// TIA Portal V16 export
// export: Created 2021-09-01T08:19:45.6334848Z, ExportSetting WithDefaults, DisplayName Totally Integrated Automation Portal, DisplayVersion V16 Update 3, DisplayName TIA Portal Version Control Interface, DisplayVersion V16 Update 2, DisplayName TIA Portal Openness, DisplayVersion V16 Update 3, DisplayName TIA Portal Teamcenter Gateway, DisplayVersion V16, DisplayName STEP 7 Professional, DisplayVersion V16 Update 3, DisplayName STEP 7 Safety, DisplayVersion V16, DisplayName WinCC Advanced, DisplayVersion V16 Update 3
TYPE "SeqStep"
// stored: IsFailsafeCompliant false
   STRUCT
      StepDev { S7_SetPoint := 'True'} : Array[1..32] of Word;
      StepDelay { S7_SetPoint := 'True'} : Array[1..32] of Time;
      initDev : Word;
      AlgN : Int;
      nStartStep { S7_SetPoint := 'True'} : Int := 1;
   END_STRUCT;
END_TYPE
